Staubli VAL3: Day10.dtx

string sInput
lists lResult
  [0]
    string sString
string sQueue
string sCorrupt
num nSum
num nCompletion
bool bCorrupt
num nResult
